// Mitsubishi GX Works2 project: EX2_Group10   PLC: FX3G

// global labels: Global1
VAR_GLOBAL
  startDay AT X007 : BOOL;
  choclateCoins AT D1100 : REAL;
  choclateContainr AT D1110 : REAL;
  nuts AT D1102 : REAL;
  nutsContainer AT D1112 : REAL;
  pictachio AT D1104 : REAL;
  pictachioContainer AT D1114 : REAL;
  kadaifHair AT D1106 : REAL;
  kadaifHairContainer AT D1116 : REAL;
  endDay AT M7 : BOOL;
  workDayLight AT Y007 : BOOL;
  emergencyButon AT X005 : BOOL;
  outOfStock AT M1 : BOOL;
  checkStock AT X004 : BOOL;
  Analog_Input1 AT D8280 : INT;
  saveAnalog AT D1200 : REAL;
END_VAR
VAR_GLOBAL CONSTANT
  constant_400 : REAL := 400.0;
END_VAR
VAR_GLOBAL
  normalizeInput AT D1202 : REAL;
END_VAR
VAR_GLOBAL CONSTANT
  constant5 : REAL := 5;
END_VAR
VAR_GLOBAL
  dubaiChoclate AT M5 : BOOL;
  mixNutsChoclate AT M6 : BOOL;
END_VAR
VAR_GLOBAL CONSTANT
  constantChoclate : REAL := 400.0;
  consant20 : REAL := 20.0;
  consant120 : REAL := 120.0;
  consant60 : REAL := 60.0;
END_VAR
VAR_GLOBAL
  picttachioContainer AT D1114 : REAL;
END_VAR
VAR_GLOBAL CONSTANT
  consant100 : REAL := 100.0;
END_VAR
VAR_GLOBAL
  startMelting AT X001 : BOOL;
  stopMelting AT X002 : BOOL;
  meltingLight AT Y001 : BOOL;
  meltingContainer AT D1118 : REAL;
  startCasting AT X003 : BOOL;
  emptyPattern AT D1204 : REAL;
  TC_1 AT TC1 : BOOL;
END_VAR
VAR_GLOBAL CONSTANT
  constant_40 : INT := 40;
END_VAR
VAR_GLOBAL
  TS_1 AT TS1 : BOOL;
  castingLight AT Y002 : BOOL;
  filling_Container AT D1206 : REAL;
  TC_6 AT TC6 : BOOL;
END_VAR
VAR_GLOBAL CONSTANT
  Const5 : INT := 50;
END_VAR
VAR_GLOBAL
  TS_6 AT TS6 : BOOL;
  TC_5 AT TC5 : BOOL;
  TS_5 AT TS5 : BOOL;
  fillingLight1 AT Y003 : BOOL;
  fillingLight4 AT Y004 : BOOL;
  castingIndicator AT M8 : BOOL;
  TC_8 AT TC8 : BOOL;
  TS_8 AT TS8 : BOOL;
  flickerIndicator AT M10 : BOOL;
  flickingIndicator AT M10 : BOOL;
END_VAR
VAR_GLOBAL CONSTANT
  Const1 : INT := 10;
END_VAR
VAR_GLOBAL
  flickingLight AT M15 : BOOL;
  flashLight AT M15 : BOOL;
  startFreezing AT X006 : BOOL;
  freezingLight AT Y006 : BOOL;
  TC_7 AT TC7 : BOOL;
END_VAR
VAR_GLOBAL CONSTANT
  Const3 : INT := 30;
END_VAR
VAR_GLOBAL
  packingSwitch AT X000 : BOOL;
  packingLight AT Y005 : BOOL;
  CC_11 AT CC11 : BOOL;
END_VAR
VAR_GLOBAL CONSTANT
  Counter4 : INT := 4;
END_VAR
VAR_GLOBAL
  CS_11 AT CS11 : BOOL;
  storage AT D1300 : REAL;
END_VAR
VAR_GLOBAL CONSTANT
  choclatePack : REAL := 1.0;
END_VAR
VAR_GLOBAL
  TS_7 AT TS7 : BOOL;
  TC_11 AT TC11 : BOOL;
  iteration AT M20 : BOOL;
  singleChocolate AT CC12 : BOOL;
END_VAR
VAR_GLOBAL CONSTANT
  Counter1 : INT := 1;
END_VAR
VAR_GLOBAL
  package AT CC13 : BOOL;
  CS_13 AT CS13 : BOOL;
  CS_12 AT CS12 : BOOL;
END_VAR
VAR_GLOBAL CONSTANT
  Counter_1 : REAL := 1.0;
END_VAR
VAR_GLOBAL
  normalizedOutput AT D1302 : REAL;
  analogOutput AT D8282 : INT;
END_VAR
VAR_GLOBAL CONSTANT
  normalFactor : REAL := 10.0;
END_VAR
VAR_GLOBAL
  checkingStock AT M16 : BOOL;
END_VAR

// task Task_01 (event TRUE, interval 0, priority 31): POU_01

PROGRAM POU_01
(* structured ladder/FBD written out as ST: instructions are called as NAME(EN, inputs, outputs); _pN, _eN, _tN stand for wires *)
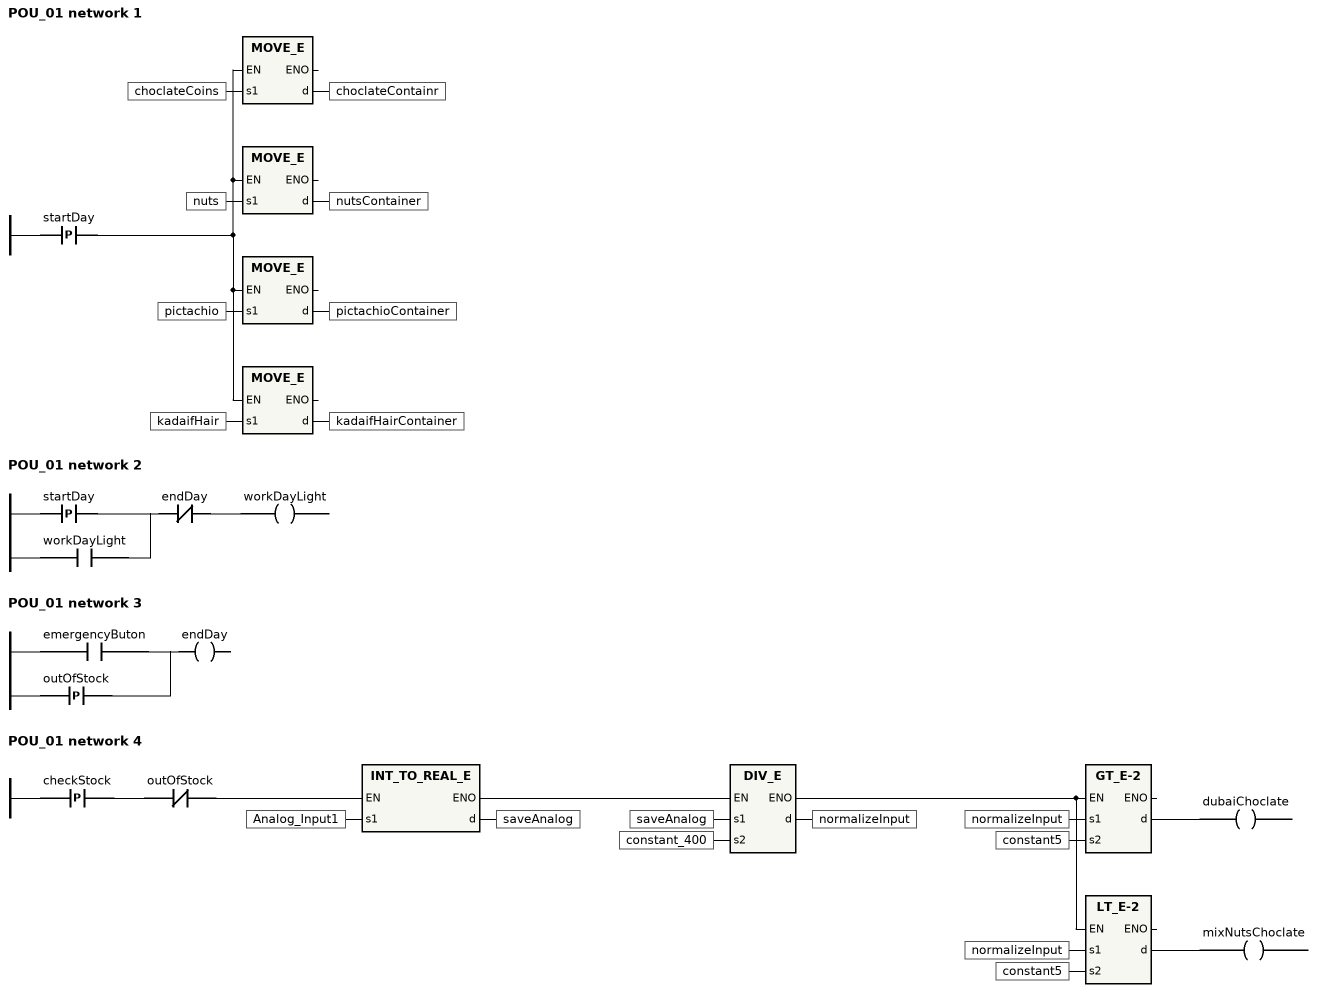
(* network 1 *)
_p1 := LDP(TRUE, startDay);
MOVE_E(_p1, choclateCoins, choclateContainr);
MOVE_E(_p1, nuts, nutsContainer);
MOVE_E(_p1, pictachio, pictachioContainer);
MOVE_E(_p1, kadaifHair, kadaifHairContainer);
(* network 2 *)
workDayLight := (LDP(TRUE, startDay) OR workDayLight) AND NOT endDay;
(* network 3 *)
endDay := emergencyButon OR LDP(TRUE, outOfStock);
(* network 4 *)
_e1 := INT_TO_REAL_E(LDP(TRUE, checkStock) AND NOT outOfStock, Analog_Input1, saveAnalog);
_e2 := DIV_E(_e1, saveAnalog, constant_400, normalizeInput);
GT_E(_e2, normalizeInput, constant5, _t3);
dubaiChoclate := _t3;
LT_E(_e2, normalizeInput, constant5, _t4);
mixNutsChoclate := _t4;
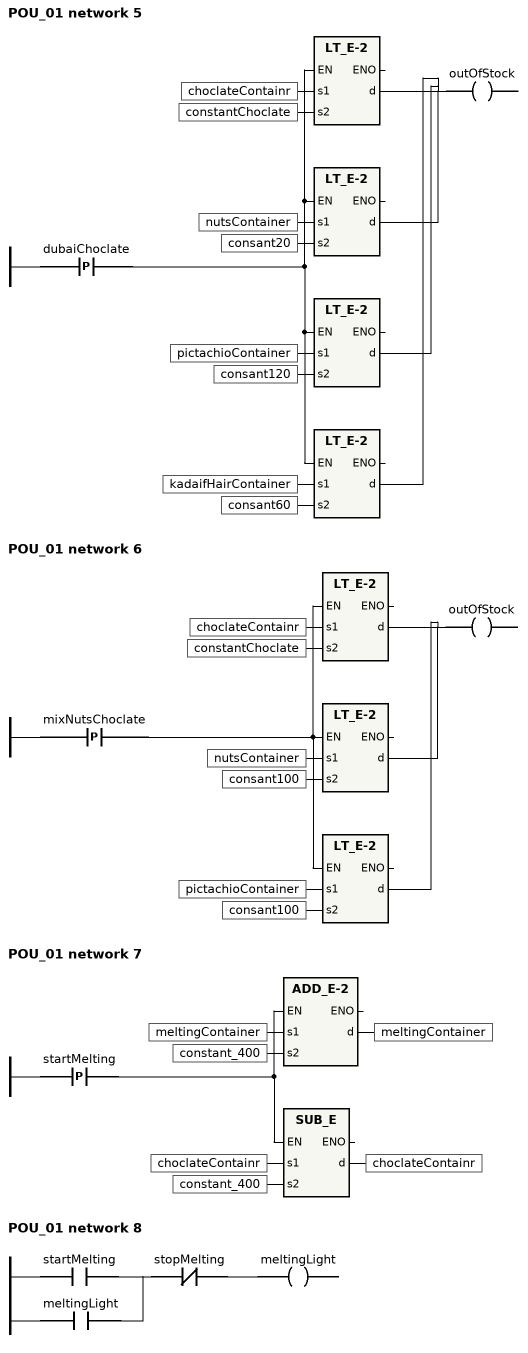
(* network 5 *)
_p1 := LDP(TRUE, dubaiChoclate);
LT_E(_p1, choclateContainr, constantChoclate, _t2);
LT_E(_p1, nutsContainer, consant20, _t3);
LT_E(_p1, pictachioContainer, consant120, _t4);
LT_E(_p1, kadaifHairContainer, consant60, _t5);
outOfStock := _t2 OR _t3 OR _t4 OR _t5;
(* network 6 *)
_p1 := LDP(TRUE, mixNutsChoclate);
LT_E(_p1, choclateContainr, constantChoclate, _t2);
LT_E(_p1, nutsContainer, consant100, _t3);
LT_E(_p1, pictachioContainer, consant100, _t4);
outOfStock := _t2 OR _t3 OR _t4;
(* network 7 *)
_p1 := LDP(TRUE, startMelting);
ADD_E(_p1, meltingContainer, constant_400, meltingContainer);
SUB_E(_p1, choclateContainr, constant_400, choclateContainr);
(* network 8 *)
meltingLight := (startMelting OR meltingLight) AND NOT stopMelting;
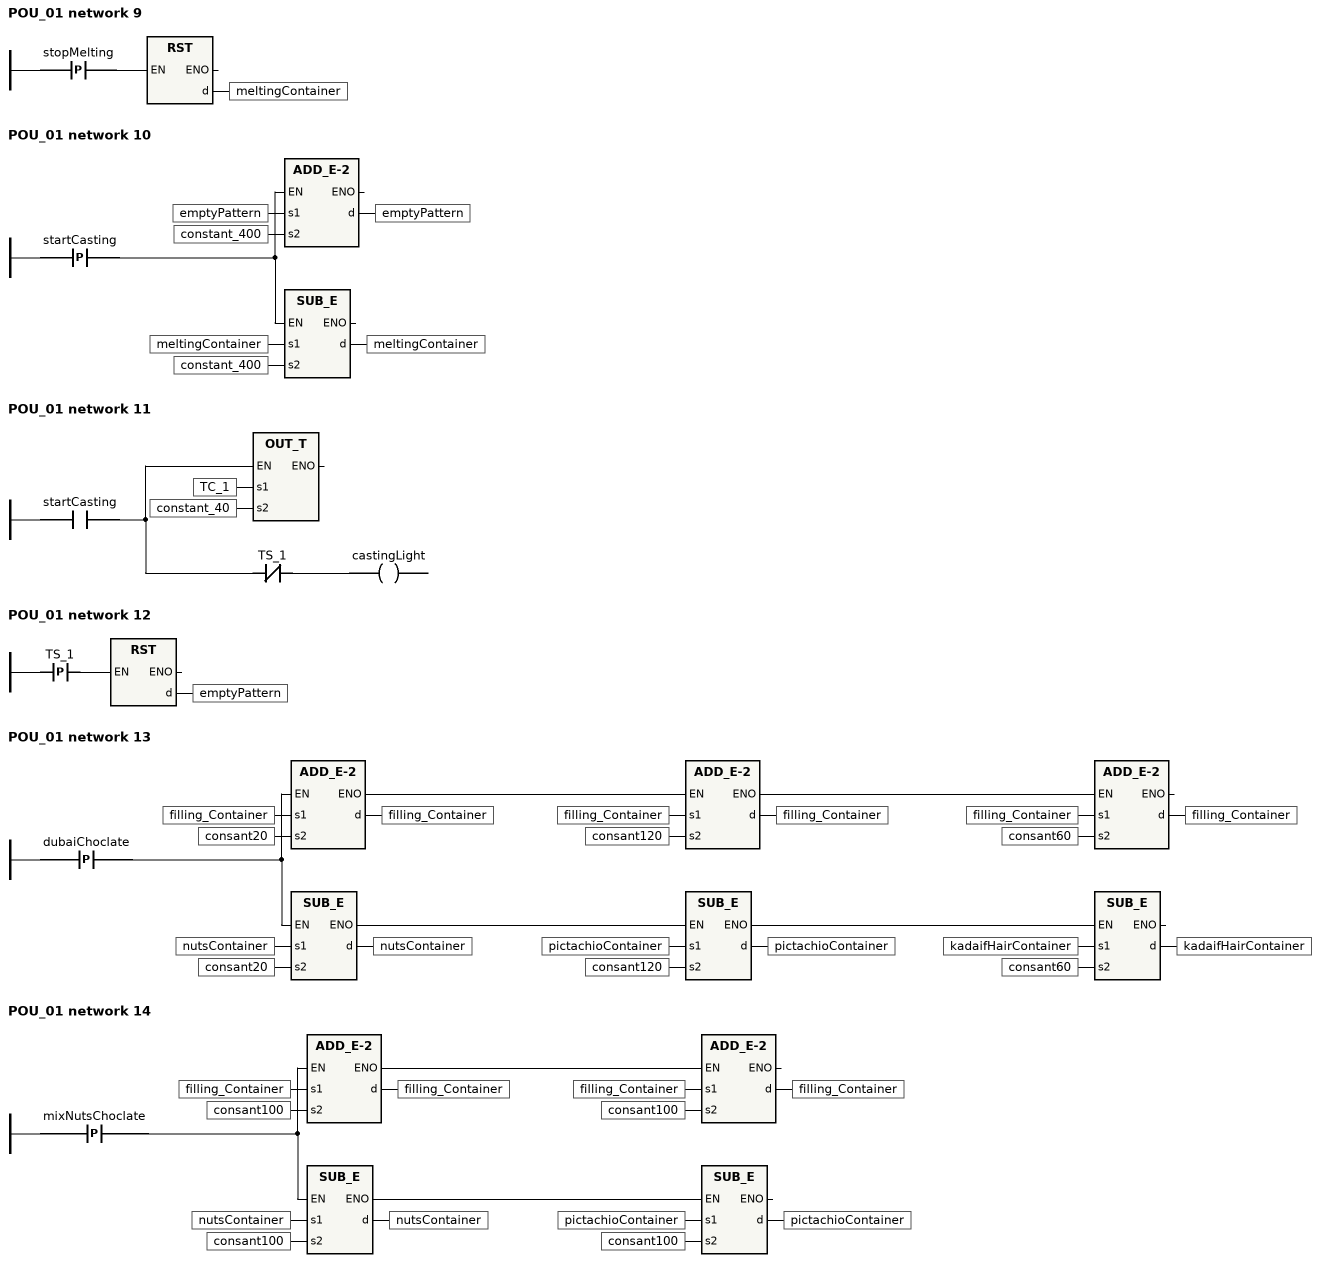
(* network 9 *)
RST(LDP(TRUE, stopMelting), meltingContainer);
(* network 10 *)
_p1 := LDP(TRUE, startCasting);
ADD_E(_p1, emptyPattern, constant_400, emptyPattern);
SUB_E(_p1, meltingContainer, constant_400, meltingContainer);
(* network 11 *)
OUT_T(startCasting, TC_1, constant_40);
castingLight := startCasting AND NOT TS_1;
(* network 12 *)
RST(LDP(TRUE, TS_1), emptyPattern);
(* network 13 *)
_p1 := LDP(TRUE, dubaiChoclate);
_e2 := ADD_E(_p1, filling_Container, consant20, filling_Container);
_e3 := ADD_E(_e2, filling_Container, consant120, filling_Container);
ADD_E(_e3, filling_Container, consant60, filling_Container);
_e4 := SUB_E(_p1, nutsContainer, consant20, nutsContainer);
_e5 := SUB_E(_e4, pictachioContainer, consant120, pictachioContainer);
SUB_E(_e5, kadaifHairContainer, consant60, kadaifHairContainer);
(* network 14 *)
_p1 := LDP(TRUE, mixNutsChoclate);
_e2 := ADD_E(_p1, filling_Container, consant100, filling_Container);
ADD_E(_e2, filling_Container, consant100, filling_Container);
_e3 := SUB_E(_p1, nutsContainer, consant100, nutsContainer);
SUB_E(_e3, pictachioContainer, consant100, pictachioContainer);
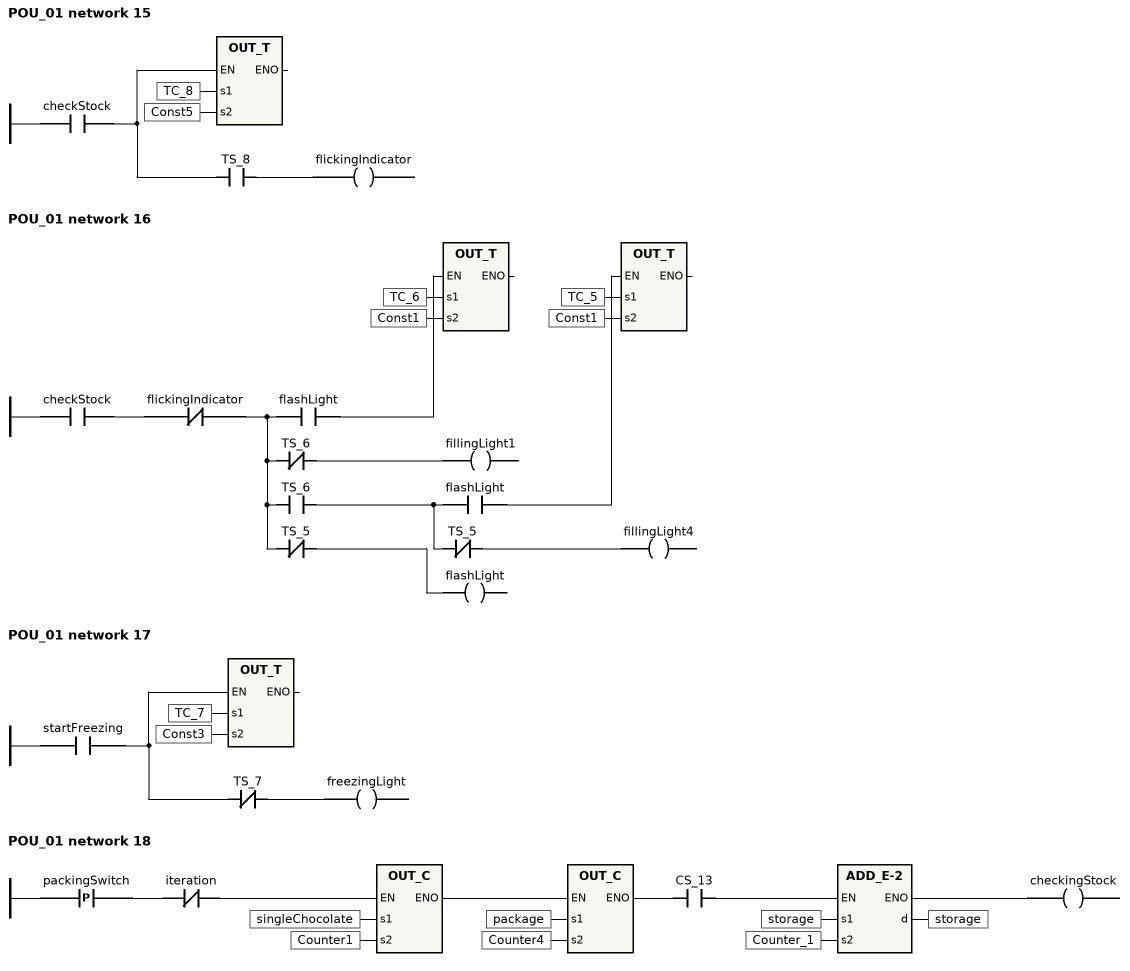
(* network 15 *)
OUT_T(checkStock, TC_8, Const5);
flickingIndicator := checkStock AND TS_8;
(* network 16 *)
_p1 := checkStock AND NOT flickingIndicator;
OUT_T(_p1 AND flashLight, TC_6, Const1);
fillingLight1 := _p1 AND NOT TS_6;
_p2 := _p1 AND TS_6;
OUT_T(_p2 AND flashLight, TC_5, Const1);
fillingLight4 := _p2 AND NOT TS_5;
flashLight := _p1 AND NOT TS_5;
(* network 17 *)
OUT_T(startFreezing, TC_7, Const3);
freezingLight := startFreezing AND NOT TS_7;
(* network 18 *)
_e1 := OUT_C(LDP(TRUE, packingSwitch) AND NOT iteration, singleChocolate, Counter1);
_e2 := OUT_C(_e1, package, Counter4);
_e3 := ADD_E(_e2 AND CS_13, storage, Counter_1, storage);
checkingStock := _e3;
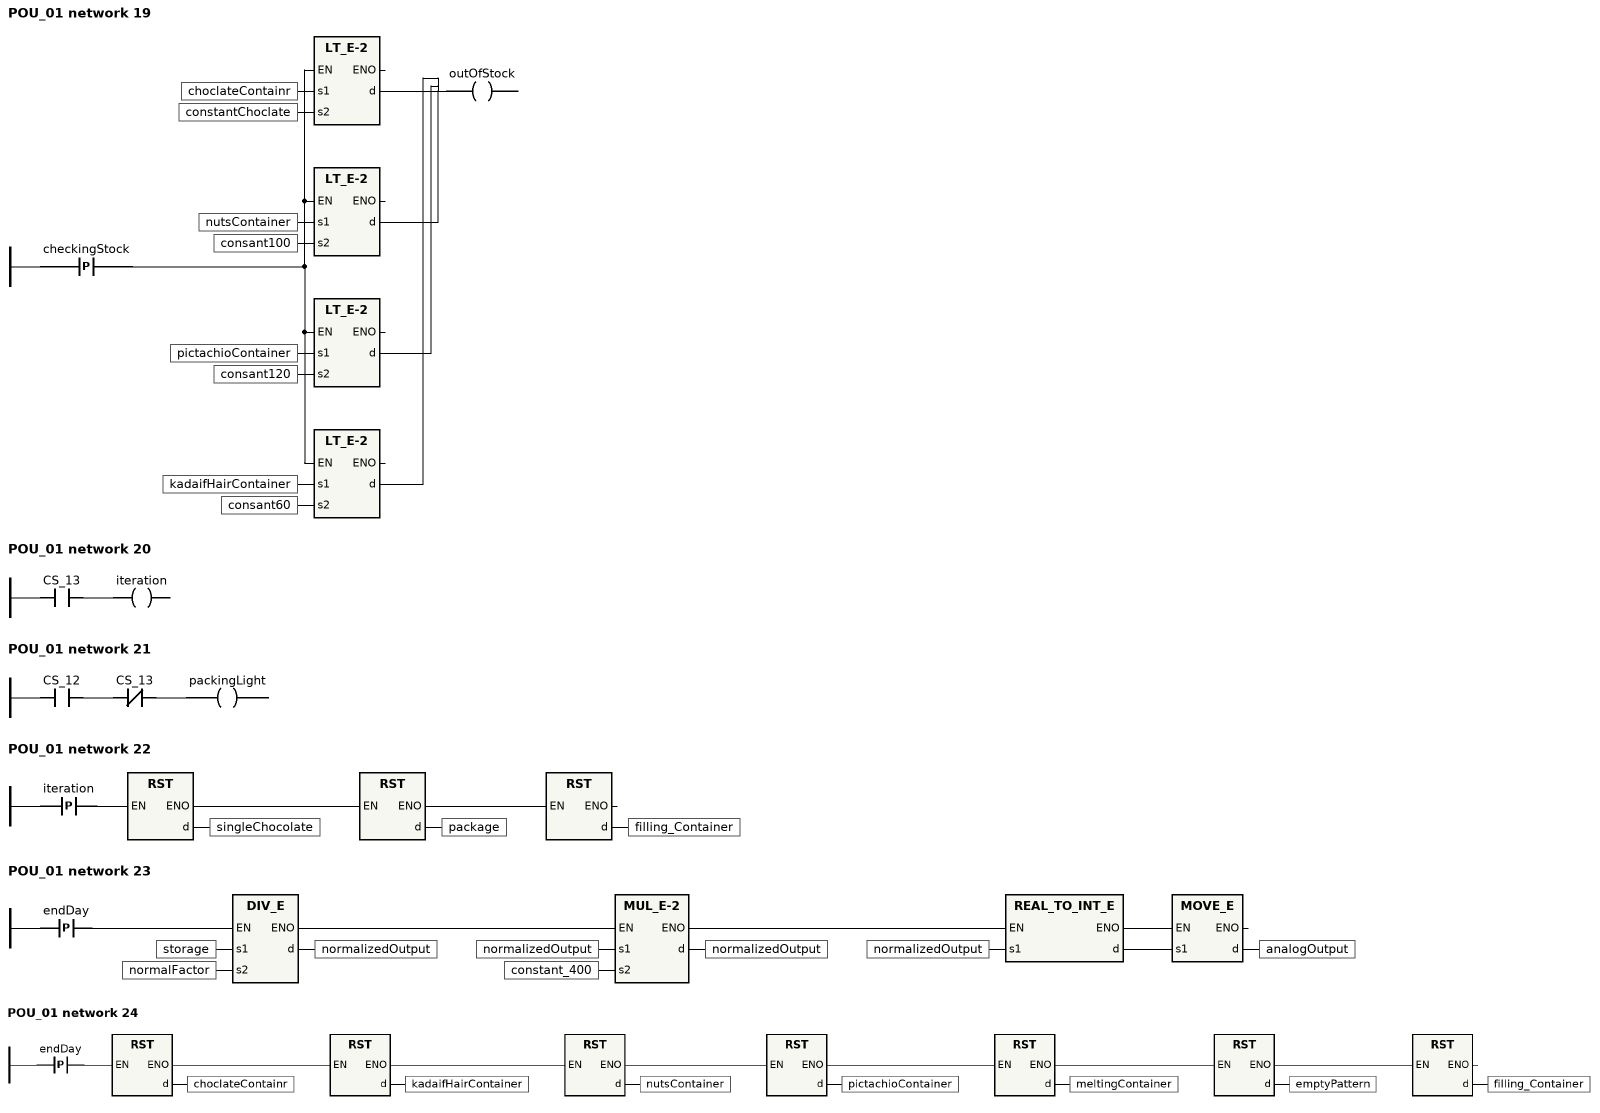
(* network 19 *)
_p1 := LDP(TRUE, checkingStock);
LT_E(_p1, choclateContainr, constantChoclate, _t2);
LT_E(_p1, nutsContainer, consant100, _t3);
LT_E(_p1, pictachioContainer, consant120, _t4);
LT_E(_p1, kadaifHairContainer, consant60, _t5);
outOfStock := _t2 OR _t3 OR _t4 OR _t5;
(* network 20 *)
iteration := CS_13;
(* network 21 *)
packingLight := CS_12 AND NOT CS_13;
(* network 22 *)
_e1 := RST(LDP(TRUE, iteration), singleChocolate);
_e2 := RST(_e1, package);
RST(_e2, filling_Container);
(* network 23 *)
_e1 := DIV_E(LDP(TRUE, endDay), storage, normalFactor, normalizedOutput);
_e2 := MUL_E(_e1, normalizedOutput, constant_400, normalizedOutput);
_e4 := REAL_TO_INT_E(_e2, normalizedOutput, _t3);
MOVE_E(_e4, _t3, analogOutput);
(* network 24 *)
_e1 := RST(LDP(TRUE, endDay), choclateContainr);
_e2 := RST(_e1, kadaifHairContainer);
_e3 := RST(_e2, nutsContainer);
_e4 := RST(_e3, pictachioContainer);
_e5 := RST(_e4, meltingContainer);
_e6 := RST(_e5, emptyPattern);
RST(_e6, filling_Container);
END_PROGRAM
